Staubli VAL3: goTo.pgx

public program goTo(tool x_tTool, mdesc x_mDesc, num x_nMoveType, bool& x_bUnreached[], num x_nIndex)
  local string l_sMessage
  local num i
  local point l_pPoint
  local joint l_jJoint
begin
  // the maximum size
  x_mDesc.blend=off
  // get the point
  call getPoint(l_pPoint,false,x_nIndex)
  //
  // step by step motion
  //
  // go to the appro
  for i=0 to size(pEditPoint.trAppro)-1
    if !pointToJoint(x_tTool,herej(),appro(l_pPoint,pEditPoint.trAppro[i]),l_jJoint)
      // not reachable
      call language:message(l_sMessage,169)
      popUpMsg(l_sMessage)
      return
    else
      if x_nMoveType==0 and i==0
        // or is not in range
        movej(appro(l_pPoint,pEditPoint.trAppro[i]),x_tTool,x_mDesc)
      else
        movel(appro(l_pPoint,pEditPoint.trAppro[i]),x_tTool,x_mDesc)
      endIf
    endIf
  endFor
  // wait to catch the point
  wait(isEmpty() or isKeyPressed(255) or cycleStatus:nWorkingStatus!=0)
  if isEmpty()
    delay(1)
    // go directly to the point is the robot is nearby the point
    if !pointToJoint(x_tTool,herej(),l_pPoint,l_jJoint)
      // not reachable
      call language:message(l_sMessage,169)
      popUpMsg(l_sMessage)
      return
    else
      movel(l_pPoint,x_tTool,x_mDesc)
      wait(isEmpty() or isKeyPressed(255) or cycleStatus:nWorkingStatus!=0)
      if isEmpty()
        delay(1)
        // go to the depart
        for i=0 to size(pEditPoint.trDepart)-1
          if !pointToJoint(x_tTool,herej(),appro(l_pPoint,pEditPoint.trDepart[i]),l_jJoint)
            // not reachable
            call language:message(l_sMessage,169)
            popUpMsg(l_sMessage)
            return
          else
            movel(appro(l_pPoint,pEditPoint.trDepart[i]),x_tTool,x_mDesc)
          endIf
        endFor
        wait(isEmpty() or isKeyPressed(255) or cycleStatus:nWorkingStatus!=0)
      endIf
    endIf
  endIf
end
